(* IEC 61131-3 sources: GradProject/, 8 files *)

(* ---- MotorController.st ---- *)
PROGRAM Test_Program
  VAR
    ESP0 AT %QX0.0 : BOOL;
  END_VAR
  VAR
    TMP : BOOL;
  END_VAR
  VAR
    TMP0 AT %QX1.3 : BOOL;
    ESP1 AT %QX0.1 : BOOL;
  END_VAR
  VAR
    TON1 : TON;
    TON2 : TON;
  END_VAR

  ESP0 := NOT(TMP) AND TMP0;
  TON1(IN := ESP0 OR ESP0, PT := T#3000ms);
  ESP1 := TON1.Q;
  TON2(IN := ESP1, PT := T#5000ms);
  TMP := TON2.Q;
END_PROGRAM

CONFIGURATION Config0

  RESOURCE Res0 ON PLC
    TASK MyTask(INTERVAL := T#50ms,PRIORITY := 0);
    PROGRAM instance0 WITH MyTask : Test_Program;
  END_RESOURCE
END_CONFIGURATION

(* ---- Test13.st ---- *)
PROGRAM Test_Program
  VAR
    ESP0 AT %QX0.0 : BOOL;
    TMP AT %IX0.3 : BOOL;
    ESP1 AT %QX0.1 : BOOL;
  END_VAR
  VAR
    TMP2 : BOOL;
    TMP4 : BOOL;
    TMP3 : BOOL;
    TON1 : TON;
    TON2 : TON;
    TON3 : TON;
  END_VAR

  ESP0 := TMP;
  TON1(IN := ESP0, PT := T#10000ms);
  ESP1 := TON1.Q;
  TON2(IN := ESP1, PT := T#10000ms);
  IF TON2.Q THEN
    ESP1 := FALSE; (*reset*)
  END_IF;
  TMP4 := NOT(TMP3);
  TON3(IN := TMP4, PT := T#30000ms);
  IF TON3.Q THEN
    ESP0 := FALSE; (*reset*)
  END_IF;
END_PROGRAM

CONFIGURATION Config0

  RESOURCE Res0 ON PLC
    TASK MyTask(INTERVAL := T#50ms,PRIORITY := 0);
    PROGRAM instance0 WITH MyTask : Test_Program;
  END_RESOURCE
END_CONFIGURATION

(* ---- Test15.st ---- *)
PROGRAM Test_Program
  VAR
    ESP0 AT %QX0.0 : BOOL;
    TMP AT %QX0.2 : BOOL;
    ESP1 AT %QX0.1 : BOOL;
  END_VAR
  VAR
    TMP2 : BOOL;
    TMP4 : BOOL;
    TMP3 : BOOL;
    TON1 : TON;
    TON2 : TON;
    TON3 : TON;
  END_VAR

  ESP0 := NOT(TMP);
  TON1(IN := ESP0, PT := T#10000ms);
  ESP1 := TON1.Q;
  TON2(IN := ESP1, PT := T#10000ms);
  IF TON2.Q THEN
    ESP1 := FALSE; (*reset*)
  END_IF;
  TMP4 := NOT(TMP3);
  TON3(IN := TMP4, PT := T#30000ms);
  IF TON3.Q THEN
    ESP0 := FALSE; (*reset*)
  END_IF;
END_PROGRAM

CONFIGURATION Config0

  RESOURCE Res0 ON PLC
    TASK MyTask(INTERVAL := T#50ms,PRIORITY := 0);
    PROGRAM instance0 WITH MyTask : Test_Program;
  END_RESOURCE
END_CONFIGURATION

(* ---- Test17.st ---- *)
PROGRAM Test_Program
  VAR
    ESP0 AT %QX0.0 : BOOL;
    TMP AT %QX0.2 : BOOL;
    ESP1 AT %QX0.1 : BOOL;
  END_VAR
  VAR
    TMP2 : BOOL;
    TMP4 : BOOL;
    TMP3 : BOOL;
    TON1 : TON;
    TON2 : TON;
  END_VAR

  ESP0 := NOT(TMP);
  TON1(IN := ESP0, PT := T#10000ms);
  ESP1 := TON1.Q;
  TON2(IN := ESP1, PT := T#10000ms);
  IF TON2.Q THEN
    ESP1 := FALSE; (*reset*)
  END_IF;
  IF ESP1 THEN
    ESP0 := FALSE; (*reset*)
  END_IF;
END_PROGRAM

CONFIGURATION Config0

  RESOURCE Res0 ON PLC
    TASK MyTask(INTERVAL := T#50ms,PRIORITY := 0);
    PROGRAM instance0 WITH MyTask : Test_Program;
  END_RESOURCE
END_CONFIGURATION

(* ---- Test24.st ---- *)
PROGRAM Test_Program
  VAR
    ESP0 AT %QX0.0 : BOOL;
  END_VAR
  VAR
    TMP : BOOL;
  END_VAR
  VAR
    ESP1 AT %QX0.1 : BOOL;
  END_VAR
  VAR
    TON1 : TON;
    TON2 : TON;
  END_VAR

  ESP0 := NOT(TMP);
  TON1(IN := ESP0, PT := T#10000ms);
  ESP1 := TON1.Q;
  TON2(IN := ESP1, PT := T#10000ms);
END_PROGRAM

CONFIGURATION Config0

  RESOURCE Res0 ON PLC
    TASK MyTask(INTERVAL := T#50ms,PRIORITY := 0);
    PROGRAM instance0 WITH MyTask : Test_Program;
  END_RESOURCE
END_CONFIGURATION

(* ---- Test25.st ---- *)
PROGRAM Test_Program
  VAR
    ESP0 AT %QX0.0 : BOOL;
  END_VAR
  VAR
    TMP : BOOL;
  END_VAR
  VAR
    ESP1 AT %QX0.1 : BOOL;
  END_VAR
  VAR
    TON1 : TON;
    TON2 : TON;
    TON0 : TON;
  END_VAR

  TON0(IN := NOT(TMP), PT := T#3000ms);
  ESP0 := TON0.Q;
  TON1(IN := ESP0 OR ESP0, PT := T#3000ms);
  ESP1 := TON1.Q;
  TON2(IN := ESP1, PT := T#5000ms);
  TMP := TON2.Q;
END_PROGRAM

CONFIGURATION Config0

  RESOURCE Res0 ON PLC
    TASK MyTask(INTERVAL := T#50ms,PRIORITY := 0);
    PROGRAM instance0 WITH MyTask : Test_Program;
  END_RESOURCE
END_CONFIGURATION

(* ---- Test26.st ---- *)
PROGRAM Test_Program
  VAR
    ESP0 AT %QX0.0 : BOOL;
    TMP AT %QX0.2 : BOOL;
    ESP1 AT %QX0.1 : BOOL;
  END_VAR
  VAR
    TON1 : TON;
    TON2 : TON;
  END_VAR

  ESP0 := TMP;
  TON1(IN := ESP0 OR ESP0, PT := T#3000ms);
  ESP1 := TON1.Q;
  TON2(IN := ESP1, PT := T#5000ms);
  TMP := TON2.Q;
END_PROGRAM

CONFIGURATION Config0

  RESOURCE Res0 ON PLC
    TASK MyTask(INTERVAL := T#50ms,PRIORITY := 0);
    PROGRAM instance0 WITH MyTask : Test_Program;
  END_RESOURCE
END_CONFIGURATION

(* ---- Test32.st ---- *)
PROGRAM Test_Program
  VAR
    ESP0 AT %QX0.0 : BOOL;
  END_VAR
  VAR
    TMP : BOOL;
  END_VAR
  VAR
    TMP0 AT %QX0.2 : BOOL;
    ESP1 AT %QX0.1 : BOOL;
  END_VAR
  VAR
    TON1 : TON;
    TON2 : TON;
  END_VAR

  ESP0 := NOT(TMP) AND TMP0;
  TON1(IN := ESP0 OR ESP0, PT := T#3000ms);
  ESP1 := TON1.Q;
  TON2(IN := ESP1, PT := T#5000ms);
  TMP := TON2.Q;
END_PROGRAM

CONFIGURATION Config0

  RESOURCE Res0 ON PLC
    TASK MyTask(INTERVAL := T#50ms,PRIORITY := 0);
    PROGRAM instance0 WITH MyTask : Test_Program;
  END_RESOURCE
END_CONFIGURATION
